// TIA Portal project "NXConnection" (V19)

(* hardware
DEVICE "S7-1500/ET200MP station_1"  S7-1500 station
   slot 0: "Rail_0"  Rack  6ES7 590-1***0-0AA0
   slot 1: "PLC_1"  CPU 1516F-3 PN/DP  6ES7 516-3FN01-0AB0  V2.6
      slot 3: "CPU display_1"  6ES7591-1BA00-0AA0
      slot 32768: "PROFINET interface_1"  X1
         slot 32769: "Port_1"  X1 P1
         slot 32770: "Port_2"  X1 P2
      slot 33024: "PROFINET interface_2"  X2
         slot 33025: "Port_1"  X2 P1
      slot 33280: "DP interface_1"  X3
   slot 2: "DI 32x24VDC HF_1"  DI 32x24VDC HF  6ES7 521-1BL00-0AB0  V2.2
   slot 3: "DQ 32x24VDC/0.5A ST_1"  DQ 32x24VDC/0.5A ST  6ES7 522-1BL00-0AB0  V2.0
   slot 4: "AI 8xU/I/RTD/TC ST_1"  AI 8xU/I/RTD/TC ST  6ES7 531-7KF00-0AB0  V2.2
   slot 5: "AQ 4xU/I ST_1"  AQ 4xU/I ST  6ES7 532-5HD00-0AB0  V2.2
DEVICE "HMI_1"  KTP700 Basic PN
   slot 0: "HMI_1"  KTP700 Basic PN  6AV2 123-2GB03-0AX0  15.1.0.0
   slot 1: "HMI_RT_1"  KTP700 Basic PN  6AV2 123-2GB03-0AX0  15.1.0.0
   slot 5: "HMI_1.IE_CP_1"  PROFINET Interface  15.0.1.0
      slot 1: "PROFINET Interface_1"  PROFINET Interface
         slot 1: "Port_1"  Port
*)

// ===== PLC "PLC_1"  CPU 1516F-3 PN/DP =====

VAR_GLOBAL   // PLC tag table "Default tag table"
   "LightSensorCube" AT %I0.0 : Bool;
   "LightSensorCylinder" AT %I0.1 : Bool;
   "LightSensorWorkpiece" AT %I0.2 : Bool;
   "LimitSwitchCylinderNotExtended" AT %I0.3 : Bool;
   "LimitSwitchCylinderRetracted" AT %I0.4 : Bool;
   "WorkpieceCylinder" AT %Q0.0 : Bool;
   "WorkpieceCube" AT %Q0.1 : Bool;
   "CylinderHeadRetract" AT %Q0.2 : Bool;
   "CylinderHeadExtend" AT %Q0.3 : Bool;
   "ConveyorLong" AT %Q0.4 : Bool;
   "ConveyorShort" AT %Q0.5 : Bool;
END_VAR

DATA_BLOCK "Main_Safety_RTG1_DB"   // DB1, F_DB
{ S7_Optimized_Access := 'TRUE' }
NAME : FUSI
VERSION : 0.1
// stored: InstanceOfName Main_Safety_RTG1
"Main_Safety_RTG1"
BEGIN
END_DATA_BLOCK

FUNCTION_BLOCK "Main_Safety_RTG1"   // FB1, F_FBD
{ S7_Optimized_Access := 'TRUE' }
BEGIN
END_FUNCTION_BLOCK

FUNCTION_BLOCK "SortingControl"   // FB2, SCL
{ S7_Optimized_Access := 'TRUE' }
VERSION : 0.1
   VAR
      "STEP" : Int;
   END_VAR
BEGIN
END_FUNCTION_BLOCK

ORGANIZATION_BLOCK "Main"   // OB1, LAD, ProgramCycle
TITLE = "Main Program Sweep (Cycle)"
{ S7_Optimized_Access := 'TRUE' }
VERSION : 0.1
   VAR_INPUT
      Initial_Call : Bool;   // Initial call of this OB
      Remanence : Bool;   // =True, if remanent data are available
   END_VAR
BEGIN
END_ORGANIZATION_BLOCK

(* ===== HMI "HMI_RT_1" =====
system functions are stored by id; their names below are inferred from use
connection "HMI_Connection_1": ETHERNET, SMART_S7_1500_OMS

HMI tags "Default tag table"
   "Tag_ScreenNumber" : UInt, internal
   "WorkpieceCube" : Bool = PLC WorkpieceCube AT %Q0.1, 1 s
   "LightSensorWorkpiece" : Bool = PLC LightSensorWorkpiece AT %I0.2, 100 ms
   "WorkpieceCylinder" : Bool = PLC WorkpieceCylinder AT %Q0.0, 1 s
   "ConveyorLong" : Bool = PLC ConveyorLong AT %Q0.4, 1 s
   "ConveyorShort" : Bool = PLC ConveyorShort AT %Q0.5, 1 s
   "CylinderHeadExtend" : Bool = PLC CylinderHeadExtend AT %Q0.3, 1 s
   "CylinderHeadRetract" : Bool = PLC CylinderHeadRetract AT %Q0.2, 1 s
   "LightSensorCylinder" : Bool = PLC LightSensorCylinder AT %I0.1, 1 s
   "LightSensorCube" : Bool = PLC LightSensorCube AT %I0.0, 1 s
   "LimitSwitchCylinderNotExtended" : Bool = PLC LimitSwitchCylinderNotExtended AT %I0.3, 1 s

Template "Template_1" 800x480
   Button "Exit" at 714,429 size 71x50; TextOff 'Exit'; PictureOff "ExitRuntime_KTP700_Basic_PN_TR"; PictureOn "ExitRuntime_KTP700_Basic_PN_TR"
      on Release: StopRuntime(0)
   Button "Template_Button" at 614,429 size 71x50; TextOff 'Text'
   Button "Template_Button_1" at 514,429 size 71x50; TextOff 'Text'
   Button "Template_Button_2" at 414,429 size 71x50; TextOff 'Text'
   Button "Template_Button_3" at 314,429 size 71x50; TextOff 'Text'
   Button "Template_Button_4" at 214,429 size 71x50; TextOff 'Text'
   Button "Alarms" at 114,429 size 71x50; TextOff 'Alarms'; PictureOff "AlarmDisplay_KTP700_Basic_PN_TR"; PictureOn "AlarmDisplay_KTP700_Basic_PN_TR"
      on Release: function_ef3f5d25("Alarm window_Unacknowledged", -1)
   Button "Start screen" at 14,429 size 71x50; TextOff 'Start screen'; PictureOff "NavigateHome_KTP700_Basic_PN_TR"; PictureOn "NavigateHome_KTP700_Basic_PN_TR"
      on Release: ActivateScreen("Root screen", 0)
   Button "Template_Button_5" at 1,52 size 71x50; TextOff 'Text'
   Button "Template_Button_6" at 1,106 size 71x50; TextOff 'Text'
   Button "Template_Button_7" at 1,159 size 71x50; TextOff 'Text'
   Button "Template_Button_8" at 1,213 size 71x50; TextOff 'Text'
   Button "Template_Button_9" at 1,267 size 71x50; TextOff 'Text'
   Button "Template_Button_10" at 1,321 size 71x50; TextOff 'Text'
   Button "Template_Button_11" at 1,374 size 71x50; TextOff 'Text'
   Button "Template_Button_12" at 727,52 size 71x50; TextOff 'Text'
   Button "Template_Button_13" at 727,106 size 71x50; TextOff 'Text'
   Button "Template_Button_14" at 727,159 size 71x50; TextOff 'Text'
   Button "Template_Button_15" at 727,213 size 71x50; TextOff 'Text'
   Button "Template_Button_16" at 727,267 size 71x50; TextOff 'Text'
   Button "Template_Button_17" at 727,321 size 71x50; TextOff 'Text'
   Button "Template_Button_18" at 727,374 size 71x50; TextOff 'Text'
   SymbolicIOField "Symbolic_IO_Field_Screen" at 93,9 size 600x33; TextOff '0'; TextOn '1'; TextList "TextList_ScreenNames"
      ProcessValue <- "Tag_ScreenNumber"
      on Change: ActivateScreenByNumber("Tag_ScreenNumber", 0)
   DateTimeField "HmiScreenItemData" at 695,25 size 105x25
   DateTimeField "HmiScreenItemData_1" at 695,0 size 105x25
   GraphicView "Logo" at 0,0 size 91x51; Picture "Logo of HMI_1"

screen "Root screen" 800x480, template "Template_1"
   on GenerateScreen: SetTag("Tag_ScreenNumber", 1)
   Button "Button_1" at 110,95 size 141x32; TextOff 'WorkpieceCube'
      on Click: InvertBit("WorkpieceCube")
   TextField "Text field_1" at 296,99 size 171x23; Text 'WorkPiece Indicator'
   Circle "Circle_1" at 486,93 size 28x28
      Appearance <- "LightSensorWorkpiece"
   Button "Button_2" at 110,140 size 161x32; TextOff 'WorkpieceCylinder'
      on Click: InvertBit("WorkpieceCylinder")
   TextField "Text field_2" at 296,144 size 164x23; Text 'WorkPiece Cylinder'
   Circle "Circle_2" at 486,138 size 28x28
      Appearance <- "LightSensorCylinder"
   Button "Button_3" at 110,185 size 141x32; TextOff 'Conveyor Long'
      on Click: InvertBit("ConveyorLong")
   TextField "Text field_3" at 296,189 size 138x23; Text 'WorkPiece Cube'
   Circle "Circle_3" at 486,183 size 28x28
      Appearance <- "LightSensorCube"
   Button "Button_4" at 110,230 size 141x32; TextOff 'Conveyor Short'
      on Click: InvertBit("ConveyorShort")
   TextField "Text field_4" at 296,234 size 137x23; Text 'Piston retracted'
   Circle "Circle_4" at 486,228 size 28x28
      Appearance <- "LimitSwitchCylinderNotExtended"
   Button "Button_5" at 110,275 size 141x32; TextOff 'Cylinder Ext'
      on Click: SetBit("CylinderHeadExtend"); ResetBit("CylinderHeadRetract")
   TextField "Text field_5" at 296,279 size 137x23; Text 'piston extended'
   Circle "Circle_5" at 486,273 size 28x28
      Appearance <- "LightSensorWorkpiece"
   Button "Button_6" at 110,327 size 141x32; TextOff 'Cylinder Ext'
      on Click: ResetBit("CylinderHeadExtend"); SetBit("CylinderHeadRetract")
*)